//==============================================================
// 14) Ramp sheet conveyor 3 speed reference
//==============================================================
instRampSheetConveyor3(
    X          := sheetConveyor3TargetSpeedMPM,
    A_UP       := MAX(0.0, machineConfig.rampAccelerationUpMPMps2),
    A_DN       := -MAX(0.0, machineConfig.rampAccelerationDownMPMps2),
    VU_MAX     := MAX(0.0, machineConfig.rampVelocityUpMaxMPMps),
    VD_MAX     := -MAX(0.0, machineConfig.rampVelocityDownMaxMPMps),
    LIMIT_HIGH := machineConfig.maximumSpeedMPM,
    LIMIT_LOW  := machineConfig.minimumSpeedMPM,
    RST        := rampReset,
    Y          => sheetConveyor3SpeedRefMPM
);


//==============================================================
// 16) Calculate real separation tracking speed using ramped references
//==============================================================
// EN: Only the real speed differential above the base speed moves the
//     separation point through the conveyors.
//     Operator speed-up is already included in base speed, so it is not
//     counted as gap opening.
sheetConveyor2OpeningSpeedMPM :=
    MAX(0.0, sheetConveyor2SpeedRefMPM - sheetConveyor2BaseSpeedMPM);

sheetConveyor3OpeningSpeedMPM :=
    MAX(0.0, sheetConveyor3SpeedRefMPM - sheetConveyor3BaseSpeedMPM);


//==============================================================
// 17) Integrate real separation tracking distance
//==============================================================
IF speedControlEnabled THEN

    IF packageSeparationState = 20 THEN

        IF sheetConveyor2OpeningSpeedMPM >= machineConfig.minimumOpeningSpeedMPM THEN

            sheetConveyor2OpeningDistanceM :=
                sheetConveyor2OpeningDistanceM +
                (sheetConveyor2OpeningSpeedMPM / 60.0) * scanTimeS;

        END_IF

    ELSIF packageSeparationState = 30 THEN

        IF sheetConveyor3OpeningSpeedMPM >= machineConfig.minimumOpeningSpeedMPM THEN

            sheetConveyor3OpeningDistanceM :=
                sheetConveyor3OpeningDistanceM +
                (sheetConveyor3OpeningSpeedMPM / 60.0) * scanTimeS;

        END_IF

    END_IF

END_IF;


//==============================================================
// 18) Publish tracking distances to outputs
//==============================================================
sheetConveyor2TrackingDistanceM := sheetConveyor2OpeningDistanceM;
sheetConveyor3TrackingDistanceM := sheetConveyor3OpeningDistanceM;
END_METHOD

//==============================================================
// SIMPLE STACKER — HMI STATUS
// EN: Maps internal status, outputs, positions and diagnostics
//     to the HMI status structure.
//==============================================================
METHOD _HmiStatus



//==============================================================
// 1) System general status
//==============================================================
hmiStatus.systemRunEnable :=
    systemRunEnable;

hmiStatus.safetyCircuitOk :=
    safetyCircuitOk;

hmiStatus.faultActive :=
    faultActive OR
    backstopFault OR
    conveyorLevelerFault OR
    sheetStackDischargeFault OR
    sheetStackDischargeConveyorFault;

hmiStatus.deviceState :=
    deviceState;


//==============================================================
// 2) Sheet conveyor group status
//==============================================================
hmiStatus.synchronizedConveyorsRunning :=
    synchronizedConveyorsRunning;

hmiStatus.sheetConveyor1Run :=
    sheetConveyor1Run;

hmiStatus.sheetConveyor2Run :=
    sheetConveyor2Run;

hmiStatus.sheetConveyor3Run :=
    sheetConveyor3Run;

hmiStatus.sheetConveyor1SpeedRefMPM :=
    sheetConveyor1SpeedRefMPM;

hmiStatus.sheetConveyor2SpeedRefMPM :=
    sheetConveyor2SpeedRefMPM;

hmiStatus.sheetConveyor3SpeedRefMPM :=
    sheetConveyor3SpeedRefMPM;

hmiStatus.syncConveyorsState :=
    syncConveyorsState;


//==============================================================
// 3) Sheet stack separation status
//==============================================================
hmiStatus.sheetStackSeparationReady :=
    sheetStackSeparationReady;

hmiStatus.sheetStackSeparationActive :=
    sheetStackSeparationActive;

hmiStatus.sheetStackBrakeActive :=
    sheetStackBrakeActive;


//==============================================================
// 4) Sheet stack discharge sequence status
//==============================================================
hmiStatus.sheetStackDischargeState :=
    sheetStackDischargeState;

hmiStatus.sheetStackDischargeStateCode :=
    sheetStackDischargeStateCode;

hmiStatus.sheetStackDischargePending :=
    sheetStackDischargePending;

hmiStatus.sheetStackDischargeActive :=
    sheetStackDischargeActive;

hmiStatus.sheetStackDischargeStarted :=
    sheetStackDischargeStarted;

hmiStatus.sheetStackDischargeFinished :=
    sheetStackDischargeFinished;

hmiStatus.sheetStackDischargeFault :=
    sheetStackDischargeFault;

hmiStatus.sheetStackDischargeFaultCode :=
    sheetStackDischargeFaultCode;

hmiStatus.sheetStackDischargeLastCycleOk :=
    sheetStackDischargeLastCycleOk;

hmiStatus.sheetStackDischargeLastResultCode :=
    sheetStackDischargeLastResultCode;

hmiStatus.sheetStackDischargeLastFaultStepCode :=
    sheetStackDischargeLastFaultStepCode;

hmiStatus.sheetStackDischargeLastFaultCode :=
    sheetStackDischargeLastFaultCode;


//==============================================================
// 5) Sheet stack discharge conveyor status
//==============================================================
hmiStatus.sheetStackDischargeConveyorState :=
    sheetStackDischargeConveyorState;

hmiStatus.sheetStackDischargeConveyorRun :=
    sheetStackDischargeConveyorRun;

hmiStatus.sheetStackDischargeConveyorSpeedRefMPM :=
    sheetStackDischargeConveyorSpeedRefMPM;

hmiStatus.sheetStackDischargeConveyorFault :=
    sheetStackDischargeConveyorFault;

hmiStatus.sheetStackDischargeConveyorFaultCode :=
    sheetStackDischargeConveyorFaultCode;


//==============================================================
// 6) Backstop status
//==============================================================
hmiStatus.backstopState :=
    backstopState;

hmiStatus.backstopHomed :=
    backstopHomed;

hmiStatus.backstopHomeRunning :=
    backstopHomeRunning;

hmiStatus.backstopInPosition :=
    backstopInPosition;

hmiStatus.backstopPositionMm :=
    backstopPositionMm;

hmiStatus.backstopTargetPositionMm :=
    backstopTargetPositionMm;

hmiStatus.backstopPositionErrorMm :=
    backstopPositionErrorMm;

hmiStatus.backstopRunFw :=
    backstopRunFw;

hmiStatus.backstopRunRev :=
    backstopRunRev;

hmiStatus.backstopSpeedRefMmps :=
    backstopSpeedRefMmps;

hmiStatus.backstopPlateUpSolenoid :=
    backstopPlateUpSolenoid;

hmiStatus.backstopSetEncoderPosition :=
    backstopSetEncoderPosition;

hmiStatus.backstopSetEncoderPositionMm :=
    backstopSetEncoderPositionMm;

hmiStatus.backstopManualInterventionActive :=
    backstopManualInterventionActive;

hmiStatus.backstopManualInterventionPositionMm :=
    backstopManualInterventionPositionMm;

hmiStatus.backstopFault :=
    backstopFault;

hmiStatus.backstopFaultCode :=
    backstopFaultCode;


//==============================================================
// 7) Conveyor leveler status
//==============================================================
hmiStatus.conveyorLevelerState :=
    conveyorLevelerState;

hmiStatus.conveyorLevelerHomed :=
    conveyorLevelerHomed;

hmiStatus.conveyorLevelerInPosition :=
    conveyorLevelerInPosition;

hmiStatus.conveyorLevelerPositionMm :=
    conveyorLevelerPositionMm;

hmiStatus.conveyorLevelerTargetPositionMm :=
    conveyorLevelerTargetPositionMm;

hmiStatus.conveyorLevelerPositionErrorMm :=
    conveyorLevelerPositionErrorMm;

hmiStatus.conveyorLevelerRunUp :=
    conveyorLevelerRunUp;

hmiStatus.conveyorLevelerRunDown :=
    conveyorLevelerRunDown;

hmiStatus.conveyorLevelerBrakeRelease :=
    conveyorLevelerBrakeRelease;

hmiStatus.conveyorLevelerSpeedRefMmps :=
    conveyorLevelerSpeedRefMmps;

hmiStatus.conveyorLevelerSetEncoderPosition :=
    conveyorLevelerSetEncoderPosition;

hmiStatus.conveyorLevelerSetEncoderPositionMm :=
    conveyorLevelerSetEncoderPositionMm;

hmiStatus.conveyorLevelerFault :=
    conveyorLevelerFault;

hmiStatus.conveyorLevelerFaultCode :=
    conveyorLevelerFaultCode;


//==============================================================
// 8) Process values
//==============================================================
hmiStatus.lineSpeedMPM :=
    lineSpeedMPM;

hmiStatus.sheetLengthMm :=
    sheetLengthMm;

hmiStatus.stackHeightMm :=
    stackHeightMm;


//==============================================================
// 9) Input / drive status mirror
//==============================================================
hmiStatus.sheetConveyor1DriveOk :=
    sheetConveyor1DriveOk;

hmiStatus.sheetConveyor2DriveOk :=
    sheetConveyor2DriveOk;

hmiStatus.sheetConveyor3DriveOk :=
    sheetConveyor3DriveOk;

hmiStatus.backstopDriveOk :=
    backstopDriveOk;

hmiStatus.conveyorLevelerDriveOk :=
    conveyorLevelerDriveOk;

hmiStatus.sheetStackDischargeConveyorDriveOk :=
    sheetStackDischargeConveyorDriveOk;
END_METHOD

METHOD _MachineAuxiliary
VAR_INPUT
END_VAR
(*



stopMachinePulse :=
    NOT safetyCircuitOk OR
    NOT sheetConveyor1DriveOk OR
    NOT sheetConveyor2DriveOk OR
    NOT sheetConveyor3DriveOk;
	NOT backstopDriveOk
	NOT conveyorLevelerDriveOk
*)
noCrushRollersUpDownValve := noCrushRollersDownCmd;

stackerRunning := systemRunEnable;


reset := resetCmd;
END_METHOD

//==============================================================
// SIMPLE STACKER — SHEET CONVEYOR GROUP CONTROL
// EN: Controls the synchronized sheet conveyor group.
//     Start/stop command latch is handled by _SystemControl().
//==============================================================
METHOD _SheetConveyorGroupControl

//==============================================================
// 1) Conditions
//==============================================================
// EN: Only synchronized sheet conveyor drives are considered here.
// PT: Apenas os inversores das esteiras sincronizadas são considerados aqui.
allSynchronizedDrivesOk :=
    sheetConveyor1DriveOk AND
    sheetConveyor2DriveOk AND
    sheetConveyor3DriveOk;


// EN: Synchronized conveyor group fault.
// PT: Falha do grupo de esteiras sincronizadas.
anyFault :=
    NOT safetyCircuitOk OR
    NOT allSynchronizedDrivesOk;

faultActive := anyFault;


//==============================================================
// 2) State machine
//==============================================================
CASE syncConveyorsState OF

    0: // IDLE
        deviceState := 'IDLE';

        sheetConveyor1Run := FALSE;
        sheetConveyor2Run := FALSE;
        sheetConveyor3Run := FALSE;

        synchronizedConveyorsRunning := FALSE;

        // EN: The group starts only when the master system is enabled
        //     and no conveyor group fault is active.
        IF systemRunEnable AND NOT anyFault THEN

            syncConveyorsState := 1;

        ELSIF systemRunEnable AND anyFault THEN

            syncConveyorsState := 10;

        END_IF


    1: // RUN
        deviceState := 'RUN';

        // EN: Outputs are also directly conditioned by systemRunEnable
        //     to avoid one-scan movement after a stop command.
        sheetConveyor1Run :=
            systemRunEnable AND
            safetyCircuitOk AND
            sheetConveyor1DriveOk;

        sheetConveyor2Run :=
            systemRunEnable AND
            safetyCircuitOk AND
            sheetConveyor2DriveOk;

        sheetConveyor3Run :=
            systemRunEnable AND
            safetyCircuitOk AND
            sheetConveyor3DriveOk;

        synchronizedConveyorsRunning :=
            sheetConveyor1Run AND
            sheetConveyor2Run AND
            sheetConveyor3Run;

        IF anyFault THEN

            syncConveyorsState := 10;

        ELSIF NOT systemRunEnable THEN

            syncConveyorsState := 0;

        END_IF


    10: // FAULT
        deviceState := 'FAULT';

        sheetConveyor1Run := FALSE;
        sheetConveyor2Run := FALSE;
        sheetConveyor3Run := FALSE;

        synchronizedConveyorsRunning := FALSE;

        // EN: Fault state is released only by reset and with all faults cleared.
        //     If systemRunEnable is still TRUE after reset, the group can start
        //     again from IDLE on the next scan.
        IF resetCmd AND NOT anyFault THEN

            syncConveyorsState := 0;

        END_IF


ELSE

    syncConveyorsState := 0;

END_CASE;
END_METHOD

//==============================================================
// SIMPLE STACKER — SHEET STACK DISCHARGE CONTROL
// EN: Controls the sheet stack discharge sequence after the sheet
//     conveyor separation cycle is completed.
//
// State code
// 0  = IDLE
// 5  = WAIT_SEPARATION
// 10 = START_DISCHARGE_POSITIONING
// 20 = WAIT_BACKSTOP_POSITION
// 30 = RUN_DISCHARGE_CONVEYOR
// 40 = START_RETURN_POSITIONING
// 50 = WAIT_BACKSTOP_RETURN
// 60 = FINISH
// 90 = ABORT_TRANSIENT
//
// Last result code
// 0 = No cycle executed yet
// 1 = Last cycle completed successfully
// 2 = Last cycle completed with manual backstop skip
// 3 = Last cycle completed/aborted by timeout
// 4 = Last cycle aborted by fault
//
// Fault code
// 0  = No fault
// 1  = Safety circuit not OK
// 2  = Sheet conveyor drive not OK
// 3  = Discharge conveyor drive/control fault
// 4  = Backstop drive/control fault
// 5  = Conveyor leveler drive/control fault
// 6  = Stacker stopped during cycle
// 10 = Wait separation timeout
// 20 = Backstop positioning timeout
// 30 = Discharge conveyor did not start timeout
// 50 = Backstop return timeout
//==============================================================
METHOD _SheetStackDischargeControl
VAR
    abortCycle : BOOL;
END_VAR


//==============================================================
// 1) Default event pulses
//==============================================================
sheetStackDischargeStarted  := FALSE;
sheetStackDischargeFinished := FALSE;


//==============================================================
// 2) Default internal requests / overrides
//==============================================================
// EN: The sequence does not write the physical discharge conveyor outputs.
//     It only generates an internal request to the conveyor control method.
sheetStackDischargeConveyorRunRequest := FALSE;

backstopTargetOverrideActive := FALSE;
backstopTargetOverridePositionMm := 0.0;

conveyorLevelerTargetOverrideActive := FALSE;
conveyorLevelerTargetOverridePositionMm := 0.0;


//==============================================================
// 3) Edge detection
//==============================================================
// EN: Separate edge detector to avoid interfering with conveyor speed control.
rPackageCompleteDischarge :=
    packageCompleteCmd AND NOT packageCompleteCmdOldDischarge;

packageCompleteCmdOldDischarge := packageCompleteCmd;


//==============================================================
// 4) Fault condition
//==============================================================
// EN: Conveyor leveler feedback is not used for sequence progress,
//     but its drive/control fault still aborts the cycle.
sheetStackDischargeFaultCondition :=
    NOT safetyCircuitOk OR
    NOT sheetConveyor1DriveOk OR
    NOT sheetConveyor2DriveOk OR
    NOT sheetConveyor3DriveOk OR
    NOT sheetStackDischargeConveyorDriveOk OR
    sheetStackDischargeConveyorFault OR
    NOT backstopDriveOk OR
    backstopFault OR
    NOT conveyorLevelerDriveOk OR
    conveyorLevelerFault;


//==============================================================
// 5) Fault code priority
//==============================================================
IF NOT safetyCircuitOk THEN

    sheetStackDischargeFaultCode := 1;

ELSIF NOT sheetConveyor1DriveOk OR
      NOT sheetConveyor2DriveOk OR
      NOT sheetConveyor3DriveOk THEN

    sheetStackDischargeFaultCode := 2;

ELSIF NOT sheetStackDischargeConveyorDriveOk OR
      sheetStackDischargeConveyorFault THEN

    sheetStackDischargeFaultCode := 3;

ELSIF NOT backstopDriveOk OR
      backstopFault THEN

    sheetStackDischargeFaultCode := 4;

ELSIF NOT conveyorLevelerDriveOk OR
      conveyorLevelerFault THEN

    sheetStackDischargeFaultCode := 5;

ELSIF NOT synchronizedConveyorsRunning THEN

    sheetStackDischargeFaultCode := 6;

END_IF;


//==============================================================
// 6) Optional reset of current sequence fault display
//==============================================================
// EN: Reset clears the current sequence fault flag,
//     but does not erase last cycle diagnostic codes.
IF resetCmd AND (sheetStackDischargeControlState = 0) THEN

    sheetStackDischargeFault := FALSE;
    sheetStackDischargeFaultCode := 0;

END_IF;


//==============================================================
// 7) Arm discharge sequence from packageCompleteCmd
//==============================================================
// EN: packageCompleteCmd is ignored if stacker is not running or if
//     any relevant drive/safety fault is active.
IF rPackageCompleteDischarge AND
   synchronizedConveyorsRunning AND
   NOT sheetStackDischargeFaultCondition AND
   NOT sheetStackDischargeActive AND
   NOT sheetStackDischargePending THEN

    sheetStackDischargePending := TRUE;

    // EN: Clear current-cycle flags when a new cycle is accepted.
    sheetStackDischargeFault := FALSE;
    sheetStackDischargeFaultCode := 0;

    sheetStackDischargeCycleHasManualSkip := FALSE;
    sheetStackDischargeCycleHasTimeout := FALSE;

END_IF;


//==============================================================
// 8) Immediate abort condition
//==============================================================
// EN: Any relevant fault during an active/pending cycle aborts the
//     sequence and automatically returns to IDLE.
//     Loss of synchronized conveyor running also aborts the cycle.
abortCycle :=
    (
        sheetStackDischargeActive OR
        sheetStackDischargePending OR
        (sheetStackDischargeControlState <> 0)
    )
    AND
    (
        sheetStackDischargeFaultCondition OR
        NOT synchronizedConveyorsRunning
    );


IF abortCycle THEN

    sheetStackDischargeConveyorRunRequest := FALSE;

    backstopTargetOverrideActive := FALSE;
    conveyorLevelerTargetOverrideActive := FALSE;

    sheetStackDischargePending := FALSE;
    sheetStackDischargeActive := FALSE;

    tonSheetStackDischarge(IN := FALSE);
    tonSheetStackDischargeStepTimeout(IN := FALSE);

    sheetStackDischargeFault := TRUE;

    sheetStackDischargeLastCycleOk := FALSE;
    sheetStackDischargeLastResultCode := 4;
    sheetStackDischargeLastFaultStepCode := sheetStackDischargeControlState;
    sheetStackDischargeLastFaultCode := sheetStackDischargeFaultCode;

    sheetStackDischargeState := 'ABORTED';
    sheetStackDischargeStateCode := 90;

    // EN: Do not clear backstopManualInterventionActive here.
    //     If the cycle aborted before return, keeping the memory is safer
    //     for the next cycle.

    // EN: No latched FAULT state. Return to IDLE automatically.
    sheetStackDischargeControlState := 0;


ELSE

    //==============================================================
    // 9) Sheet stack discharge state machine
    //==============================================================
    CASE sheetStackDischargeControlState OF

        0: // IDLE
            sheetStackDischargeState := 'IDLE';
            sheetStackDischargeStateCode := 0;

            sheetStackDischargeActive := FALSE;

            sheetStackDischargeConveyorRunRequest := FALSE;

            backstopTargetOverrideActive := FALSE;
            conveyorLevelerTargetOverrideActive := FALSE;

            tonSheetStackDischarge(IN := FALSE);
            tonSheetStackDischargeStepTimeout(IN := FALSE);

            IF sheetStackDischargePending THEN

                tonSheetStackDischarge(IN := FALSE);
                tonSheetStackDischargeStepTimeout(IN := FALSE);

                sheetStackDischargeControlState := 5;

            END_IF


        5: // WAIT_SEPARATION
            sheetStackDischargeState := 'WAIT_SEPARATION';
            sheetStackDischargeStateCode := 5;

            sheetStackDischargeActive := FALSE;

            sheetStackDischargeConveyorRunRequest := FALSE;

            backstopTargetOverrideActive := FALSE;
            conveyorLevelerTargetOverrideActive := FALSE;

            tonSheetStackDischarge(IN := FALSE);

            // EN: Wait for conveyor speed control to finish sheet stack separation.
            tonSheetStackDischargeStepTimeout(
                IN := TRUE,
                PT := machineConfig.sheetStackDischargeWaitSeparationTimeout
            );

            IF sheetStackSeparationFinished THEN

                tonSheetStackDischargeStepTimeout(IN := FALSE);

                sheetStackDischargeControlState := 10;


            ELSIF tonSheetStackDischargeStepTimeout.Q THEN

                // EN: Separation did not finish. Do not discharge.
                tonSheetStackDischargeStepTimeout(IN := FALSE);

                sheetStackDischargePending := FALSE;
                sheetStackDischargeActive := FALSE;

                sheetStackDischargeFault := TRUE;
                sheetStackDischargeFaultCode := 10;

                sheetStackDischargeLastCycleOk := FALSE;
                sheetStackDischargeLastResultCode := 3;
                sheetStackDischargeLastFaultStepCode := 5;
                sheetStackDischargeLastFaultCode := 10;

                sheetStackDischargeControlState := 0;

            END_IF


        10: // START_DISCHARGE_POSITIONING
            sheetStackDischargeState := 'START_POSITIONING';
            sheetStackDischargeStateCode := 10;

            sheetStackDischargePending := FALSE;
            sheetStackDischargeActive := TRUE;
            sheetStackDischargeStarted := TRUE;

            tonSheetStackDischarge(IN := FALSE);
            tonSheetStackDischargeStepTimeout(IN := FALSE);

            //======================================================
            // EN: Latch programmed backstop target for this cycle.
            //     This is the normal position based on sheet length.
            //======================================================
            backstopProgrammedDischargeTargetMm :=
                LIMIT(
                    machineConfig.backstopMinPositionMm,
                    MAX(0.0, sheetLengthMm) +
                        machineConfig.backstopSheetLengthOffsetMm,
                    machineConfig.backstopMaxPositionMm
                );

            //======================================================
            // EN: Define safe opening base position.
            //
            // If the operator manually moved the backstop before the
            // automatic cycle, use the greater value between:
            // - programmed position
            // - last manual intervention position
            //
            // This prevents the automatic opening override from closing
            // the backstop onto the material.
            //
            // If there was no manual intervention, use only the programmed
            // position as the base.
            //======================================================
            IF backstopManualInterventionActive THEN

                backstopDischargeOpenBasePositionMm :=
                    MAX(
                        backstopProgrammedDischargeTargetMm,
                        backstopManualInterventionPositionMm
                    );

            ELSE

                backstopDischargeOpenBasePositionMm :=
                    backstopProgrammedDischargeTargetMm;

            END_IF;

            //======================================================
            // EN: Latch safe discharge open target.
            //     Offset is applied after selecting the safe base.
            //======================================================
            backstopDischargeOpenTargetMm :=
                LIMIT(
                    machineConfig.backstopMinPositionMm,
                    backstopDischargeOpenBasePositionMm +
                        machineConfig.backstopDischargeOpenOffsetMm,
                    machineConfig.backstopMaxPositionMm
                );

            // EN: Request safe backstop opening.
            //     Backstop control accepts it only in auto.
            backstopTargetOverrideActive := TRUE;
            backstopTargetOverridePositionMm := backstopDischargeOpenTargetMm;

            // EN: Request conveyor leveler to move up.
            //     The sequence does not wait for leveler feedback.
            conveyorLevelerTargetOverrideActive := TRUE;
            conveyorLevelerTargetOverridePositionMm :=
                machineConfig.conveyorLevelerMaxPositionMm;

            sheetStackDischargeControlState := 20;


        20: // WAIT_BACKSTOP_POSITION
            sheetStackDischargeState := 'WAIT_BACKSTOP_POSITION';
            sheetStackDischargeStateCode := 20;

            sheetStackDischargeActive := TRUE;

            // EN: Keep safe latched backstop discharge target active.
            backstopTargetOverrideActive := TRUE;
            backstopTargetOverridePositionMm := backstopDischargeOpenTargetMm;

            // EN: Keep conveyor leveler up target active.
            //     Feedback is intentionally ignored for sequence progress.
            conveyorLevelerTargetOverrideActive := TRUE;
            conveyorLevelerTargetOverridePositionMm :=
                machineConfig.conveyorLevelerMaxPositionMm;

            // EN: If backstop is not in auto, do not wait for it.
            IF NOT backstopAutoCmd THEN

                sheetStackDischargeCycleHasManualSkip := TRUE;

                tonSheetStackDischargeStepTimeout(IN := FALSE);

                sheetStackDischargeControlState := 30;


            ELSIF backstopInPosition THEN

                tonSheetStackDischargeStepTimeout(IN := FALSE);

                sheetStackDischargeControlState := 30;


            ELSE

                tonSheetStackDischargeStepTimeout(
                    IN := TRUE,
                    PT := machineConfig.sheetStackDischargePositioningTimeout
                );

                IF tonSheetStackDischargeStepTimeout.Q THEN

                    // EN: Do not stay trapped waiting for backstop.
                    //     Continue the cycle, but record timeout diagnostic.
                    tonSheetStackDischargeStepTimeout(IN := FALSE);

                    sheetStackDischargeCycleHasTimeout := TRUE;

                    sheetStackDischargeFault := TRUE;
                    sheetStackDischargeFaultCode := 20;

                    sheetStackDischargeLastCycleOk := FALSE;
                    sheetStackDischargeLastResultCode := 3;
                    sheetStackDischargeLastFaultStepCode := 20;
                    sheetStackDischargeLastFaultCode := 20;

                    sheetStackDischargeControlState := 30;

                END_IF

            END_IF


        30: // RUN_DISCHARGE_CONVEYOR
            sheetStackDischargeState := 'DISCHARGING';
            sheetStackDischargeStateCode := 30;

            sheetStackDischargeActive := TRUE;

            // EN: Keep safe latched backstop discharge target active
            //     while discharging.
            backstopTargetOverrideActive := TRUE;
            backstopTargetOverridePositionMm := backstopDischargeOpenTargetMm;

            // EN: Keep conveyor leveler up while discharging.
            conveyorLevelerTargetOverrideActive := TRUE;
            conveyorLevelerTargetOverridePositionMm :=
                machineConfig.conveyorLevelerMaxPositionMm;

            // EN: Request discharge conveyor run.
            //     Physical output is controlled by _SheetStackDischargeConveyorControl.
            sheetStackDischargeConveyorRunRequest := TRUE;

            // EN: If conveyor is not actually running, use start timeout.
            IF NOT sheetStackDischargeConveyorRun THEN

                tonSheetStackDischarge(IN := FALSE);

                tonSheetStackDischargeStepTimeout(
                    IN := TRUE,
                    PT := machineConfig.sheetStackDischargeConveyorStartTimeout
                );

                IF tonSheetStackDischargeStepTimeout.Q THEN

                    // EN: Conveyor did not start. Do not stay trapped.
                    tonSheetStackDischargeStepTimeout(IN := FALSE);

                    sheetStackDischargeConveyorRunRequest := FALSE;

                    sheetStackDischargeCycleHasTimeout := TRUE;

                    sheetStackDischargeFault := TRUE;
                    sheetStackDischargeFaultCode := 30;

                    sheetStackDischargeLastCycleOk := FALSE;
                    sheetStackDischargeLastResultCode := 3;
                    sheetStackDischargeLastFaultStepCode := 30;
                    sheetStackDischargeLastFaultCode := 30;

                    sheetStackDischargeControlState := 40;

                END_IF


            ELSE

                // EN: Conveyor is running. Count real discharge time.
                tonSheetStackDischargeStepTimeout(IN := FALSE);

                tonSheetStackDischarge(
                    IN := TRUE,
                    PT := machineConfig.sheetStackDischargeTime
                );

                IF tonSheetStackDischarge.Q THEN

                    tonSheetStackDischarge(IN := FALSE);

                    sheetStackDischargeConveyorRunRequest := FALSE;

                    sheetStackDischargeControlState := 40;

                END_IF

            END_IF


        40: // START_RETURN_POSITIONING
            sheetStackDischargeState := 'START_RETURN';
            sheetStackDischargeStateCode := 40;

            sheetStackDischargeActive := TRUE;

            sheetStackDischargeConveyorRunRequest := FALSE;

            tonSheetStackDischarge(IN := FALSE);
            tonSheetStackDischargeStepTimeout(IN := FALSE);

            // EN: Request backstop return to the latched programmed target.
            //     The override remains active until the backstop returns.
            backstopTargetOverrideActive := TRUE;
            backstopTargetOverridePositionMm :=
                backstopProgrammedDischargeTargetMm;

            // EN: Request conveyor leveler to return down.
            //     The sequence does not wait for leveler feedback.
            conveyorLevelerTargetOverrideActive := TRUE;
            conveyorLevelerTargetOverridePositionMm :=
                machineConfig.conveyorLevelerMinPositionMm;

            sheetStackDischargeControlState := 50;


        50: // WAIT_BACKSTOP_RETURN
            sheetStackDischargeState := 'WAIT_BACKSTOP_RETURN';
            sheetStackDischargeStateCode := 50;

            sheetStackDischargeActive := TRUE;

            sheetStackDischargeConveyorRunRequest := FALSE;

            // EN: Keep backstop return target active.
            backstopTargetOverrideActive := TRUE;
            backstopTargetOverridePositionMm :=
                backstopProgrammedDischargeTargetMm;

            // EN: Keep conveyor leveler return target active.
            //     Feedback is intentionally ignored for sequence progress.
            conveyorLevelerTargetOverrideActive := TRUE;
            conveyorLevelerTargetOverridePositionMm :=
                machineConfig.conveyorLevelerMinPositionMm;

            // EN: If backstop is not in auto, do not wait for it.
            IF NOT backstopAutoCmd THEN

                sheetStackDischargeCycleHasManualSkip := TRUE;

                tonSheetStackDischargeStepTimeout(IN := FALSE);

                sheetStackDischargeControlState := 60;


            ELSIF backstopInPosition THEN

                tonSheetStackDischargeStepTimeout(IN := FALSE);

                sheetStackDischargeControlState := 60;


            ELSE

                tonSheetStackDischargeStepTimeout(
                    IN := TRUE,
                    PT := machineConfig.sheetStackDischargeReturnTimeout
                );

                IF tonSheetStackDischargeStepTimeout.Q THEN

                    // EN: Do not stay trapped waiting for return.
                    tonSheetStackDischargeStepTimeout(IN := FALSE);

                    sheetStackDischargeCycleHasTimeout := TRUE;

                    sheetStackDischargeFault := TRUE;
                    sheetStackDischargeFaultCode := 50;

                    sheetStackDischargeLastCycleOk := FALSE;
                    sheetStackDischargeLastResultCode := 3;
                    sheetStackDischargeLastFaultStepCode := 50;
                    sheetStackDischargeLastFaultCode := 50;

                    sheetStackDischargeControlState := 60;

                END_IF

            END_IF


        60: // FINISH
            sheetStackDischargeState := 'FINISH';
            sheetStackDischargeStateCode := 60;

            sheetStackDischargeActive := FALSE;
            sheetStackDischargePending := FALSE;
            sheetStackDischargeFinished := TRUE;

            sheetStackDischargeConveyorRunRequest := FALSE;

            backstopTargetOverrideActive := FALSE;
            conveyorLevelerTargetOverrideActive := FALSE;

            tonSheetStackDischarge(IN := FALSE);
            tonSheetStackDischargeStepTimeout(IN := FALSE);

            IF sheetStackDischargeCycleHasTimeout THEN

                sheetStackDischargeLastCycleOk := FALSE;
                sheetStackDischargeLastResultCode := 3;

                // EN: Keep manual intervention memory after timeout.
                //     The backstop may not have returned correctly.

            ELSIF sheetStackDischargeCycleHasManualSkip THEN

                sheetStackDischargeLastCycleOk := FALSE;
                sheetStackDischargeLastResultCode := 2;
                sheetStackDischargeLastFaultStepCode := 0;
                sheetStackDischargeLastFaultCode := 0;

                sheetStackDischargeFault := FALSE;
                sheetStackDischargeFaultCode := 0;

                // EN: Keep manual intervention memory because the backstop
                //     was not controlled automatically.


            ELSE

                sheetStackDischargeLastCycleOk := TRUE;
                sheetStackDischargeLastResultCode := 1;
                sheetStackDischargeLastFaultStepCode := 0;
                sheetStackDischargeLastFaultCode := 0;

                sheetStackDischargeFault := FALSE;
                sheetStackDischargeFaultCode := 0;

                // EN: Cycle completed correctly and backstop returned to
                //     programmed target. Clear manual intervention memory.
                backstopManualInterventionActive := FALSE;
                backstopManualInterventionPositionMm := 0.0;

            END_IF

            // EN: Always return to IDLE automatically.
            sheetStackDischargeControlState := 0;


    ELSE

        sheetStackDischargeControlState := 0;

    END_CASE;

END_IF;
END_METHOD

//==============================================================
// SIMPLE STACKER — SHEET STACK DISCHARGE CONVEYOR CONTROL
// EN: Controls the sheet stack discharge conveyor.
//     Conveyor runs while manual button is pressed or while
//     automatic request is active and conveyor automatic mode is enabled.
//
// Fault code
// 0 = No fault
// 1 = Safety circuit not OK
// 2 = Discharge conveyor drive not OK
//==============================================================
METHOD _SheetStackDischargeConveyorControl
VAR
    manualRunRequest   : BOOL;
    automaticRunRequest: BOOL;
    finalRunRequest    : BOOL;
END_VAR
//==============================================================
// SIMPLE STACKER — SHEET STACK DISCHARGE CONVEYOR CONTROL
// EN: Controls the sheet stack discharge conveyor in manual pulse
//     or automatic sequence request.
//==============================================================


//==============================================================
// 1) Default outputs
//==============================================================
sheetStackDischargeConveyorRun := FALSE;
sheetStackDischargeConveyorSpeedRefMPM := 0.0;


//==============================================================
// 2) Run request selection
//==============================================================
// EN: Manual command is momentary. Conveyor runs while button is pressed.
manualRunRequest :=
    sheetStackDischargeConveyorManualRunCmd;


// EN: Automatic request is generated by the discharge sequence.
//     This conveyor is assumed to be available for automatic cycle
//     whenever the master system is enabled.
automaticRunRequest :=
    sheetStackDischargeConveyorRunRequest;


// EN: Master system enable blocks both manual and automatic movement.
finalRunRequest :=
    systemRunEnable AND
    (
        manualRunRequest OR
        automaticRunRequest OR
		backstopHomeRunning
    );


//==============================================================
// 3) Fault detection
//==============================================================
IF NOT safetyCircuitOk THEN

    sheetStackDischargeConveyorState := 'SAFETY_OFF';

    sheetStackDischargeConveyorFault := TRUE;
    sheetStackDischargeConveyorFaultCode := 1;


ELSIF NOT sheetStackDischargeConveyorDriveOk THEN

    sheetStackDischargeConveyorState := 'DRIVE_NOT_OK';

    sheetStackDischargeConveyorFault := TRUE;
    sheetStackDischargeConveyorFaultCode := 2;


ELSE

    //==============================================================
    // 4) Fault reset
    //==============================================================
    IF resetCmd THEN

        sheetStackDischargeConveyorFault := FALSE;
        sheetStackDischargeConveyorFaultCode := 0;

    END_IF;


    //==============================================================
    // 5) Conveyor output control
    //==============================================================
    IF sheetStackDischargeConveyorFault THEN

        sheetStackDischargeConveyorState := 'FAULT';

        sheetStackDischargeConveyorRun := FALSE;
        sheetStackDischargeConveyorSpeedRefMPM := 0.0;


    ELSIF NOT systemRunEnable THEN

        // EN: Master stop disables movement without generating a conveyor fault.
        sheetStackDischargeConveyorState := 'SYSTEM_DISABLED';

        sheetStackDischargeConveyorRun := FALSE;
        sheetStackDischargeConveyorSpeedRefMPM := 0.0;


    ELSIF finalRunRequest THEN

        IF automaticRunRequest THEN

            sheetStackDischargeConveyorState := 'AUTO_RUN';

        ELSE

            sheetStackDischargeConveyorState := 'MANUAL_RUN';

        END_IF;

        sheetStackDischargeConveyorRun := TRUE;

        sheetStackDischargeConveyorSpeedRefMPM :=
            LIMIT(
                0.0,
                machineConfig.sheetStackDischargeConveyorSpeedMPM,
                machineConfig.maximumSpeedMPM
            );


    ELSE

        sheetStackDischargeConveyorState := 'STOP';

        sheetStackDischargeConveyorRun := FALSE;
        sheetStackDischargeConveyorSpeedRefMPM := 0.0;

    END_IF

END_IF;
END_METHOD

//==============================================================
// SIMPLE STACKER — SYSTEM CONTROL
// EN: Master system run enable and automatic homing requests.
//==============================================================
METHOD _SystemControl

//==============================================================
// 1) Edge detection
//==============================================================
rStartCmd := startCmd AND NOT startCmdOld;
startCmdOld := startCmd;

rStopCmd := stopCmd AND NOT stopCmdOld;
stopCmdOld := stopCmd;



//==============================================================
// 2) Stop machine pulse on critical fault
//==============================================================
stopMachineFaultCondition :=
    NOT safetyCircuitOk OR
    NOT sheetConveyor1DriveOk OR
    NOT sheetConveyor2DriveOk OR
    NOT sheetConveyor3DriveOk OR
    NOT backstopDriveOk OR
    NOT conveyorLevelerDriveOk OR
    NOT sheetStackDischargeConveyorDriveOk;

rStopMachineFaultCondition :=
    stopMachineFaultCondition AND
    NOT stopMachineFaultConditionOld;

stopMachineFaultConditionOld :=
    stopMachineFaultCondition;

tpStopMachinePulse(
    IN := rStopMachineFaultCondition,
    PT := T#500MS
);

stopMachinePulse :=
    tpStopMachinePulse.Q;


//==============================================================
// 2) Default one-scan requests
//==============================================================
backstopAutoHomeRequest := FALSE;
conveyorLevelerAutoHomeRequest := FALSE;


//==============================================================
// 3) Master system run enable
//==============================================================
IF NOT safetyCircuitOk THEN

    systemRunEnable := FALSE;

ELSIF rStopCmd THEN

    systemRunEnable := FALSE;

ELSIF rStartCmd THEN

    systemRunEnable := TRUE;

END_IF;


//==============================================================
// 4) Automatic homing on system start
//==============================================================
// EN: Auto-home is generated only on the rising edge of startCmd.
//     Each axis must be enabled in automatic mode.
//     This prevents automatic movement of axes intentionally left in manual.
IF rStartCmd AND systemRunEnable THEN

    // Backstop auto-home
    IF backstopAutoCmd AND
       NOT backstopHomed AND
       NOT backstopFault THEN

        backstopAutoHomeRequest := TRUE;

    END_IF;


    // Conveyor leveler auto-home
    IF conveyorLevelerAutoCmd AND
       NOT conveyorLevelerHomed AND
       NOT conveyorLevelerFault THEN

        conveyorLevelerAutoHomeRequest := TRUE;

    END_IF;

END_IF;
END_METHOD

END_FUNCTION_BLOCK

(* stored: Version 1.1.0.1
   POU FB_SimpleSheetStackerControl_2: Id {a7ba3e84-122c-47b4-abea-ae2258a62e15}, SpecialFunc None
   Method _AlarmControl: Id {6d7e5915-5951-4568-9311-0f0d827bd932}
   Method _BackstopControl: Id {4630acca-839a-4e96-8b98-58296d48f85a}
   Method _ConveyorLevelerControl: Id {55437bf2-fc0d-4f35-ba84-26edd1ad683b}
   Method _ConveyorSpeedControl: Id {da00ad84-56bf-462f-9e06-eff32affd7c5}
   Method _HmiStatus: Id {f9477d37-9147-4faa-9138-fe68d9f4b06c}
   Method _MachineAuxiliary: Id {60af832d-e497-48ee-9a7d-b8fbcb9c54a5}
   Method _SheetConveyorGroupControl: Id {947708c5-924b-413f-b733-e8ba8150010a}
   Method _SheetStackDischargeControl: Id {175af176-0d4d-46cc-b480-83d48d813a4a}
   Method _SheetStackDischargeConveyorControl: Id {dcf53f48-bceb-4e44-8299-325280c97506}
   Method _SystemControl: Id {e5f398cc-9a83-4964-ae94-2dbddd399242} *)
